// TIA Portal project "CHD" (V17)

(* hardware
DEVICE "HMI_1"  KTP400 Comfort
   slot 0: "HMI_1"  KTP400 Comfort  6AV2 124-2DC01-0AX0  17.0.0.0
   slot 1: "HMI_RT_1"  KTP400 Comfort  6AV2 124-2DC01-0AX0  17.0.0.0
   slot 5: "HMI_1.IE_CP_1"  PROFINET Interface  17.0.0.0
      slot 1: "PROFINET Interface_1"  PROFINET Interface
         slot 1: "Port_1"  Port
   slot 7: "HMI_1.MPI/DP_CP_1"  MPI/DP Interface  17.0.0.0
DEVICE "S7-1200 station_1"  S7-1200 Station
   slot 0: "Rack_0"  S7-1200 Rack  Rack  V1.0
   slot 1: "PLC_1"  CPU 1211C DC/DC/Rly  6ES7 211-1HE40-0XB0  V4.3
*)

// ===== PLC "PLC_1"  CPU 1211C DC/DC/Rly =====

ORGANIZATION_BLOCK "Main"   // OB1, LAD, ProgramCycle
TITLE = "Main Program Sweep (Cycle)"
{ S7_Optimized_Access := 'TRUE' }
VERSION : 0.1
   VAR_INPUT
      Initial_Call : Bool;   // Initial call of this OB
      Remanence : Bool;   // =True, if remanent data are available
   END_VAR
BEGIN
END_ORGANIZATION_BLOCK

(* ===== HMI "HMI_RT_1" =====
connection "HMI_Connection_1": ETHERNET, S7_1200_OMS

HMI tags "Default tag table"
   "HMI_Tag_1" : Bool = PLC "BP Marche" AT %I0.1, 1 s

Template "Template_1" 480x272
   Button "Template_Button" at 415,70 size 63x63; TextOff 'Text'
   Button "Template_Button_1" at 415,138 size 63x63; TextOff 'Text'
   Button "Template_Button_2" at 415,207 size 63x63; TextOff 'Text'
   Button "Template_Button_3" at 415,1 size 63x63; TextOff 'Text'

screen "Root screen" 480x272, template "Template_1"
   Circle "Circle_1" at 102,67 size 112x112
      Appearance <- "HMI_Tag_1"
*)